{attribute 'Tc2GvlVarNames'}
VAR_CONFIG
END_VAR

(* stored: Version 1.1.0.1, ProductVersion 3.1.4020.12
   GVL Variablen_Konfiguration: Id {b8ec1b48-9aba-4587-aab5-2261518ee68e} *)
